// TIA Portal V18 export
DATA_BLOCK "CS_Drive_PL"   // DB10, Motion_DB
// stored: InstanceOfName TO_SynchronousAxis, OfSystemLibElement TO_SynchronousAxis, OfSystemLibVersion 7.0
TO_SynchronousAxis   // technology object, version 7.0
// stored: Connection Interface Actor, InputAddress 400, OutputAddress 400
// stored: Connection Interface Sensor[1], InputAddress 400, OutputAddress 400, SensorIndexInActorTelegram 1
   // // inherited from TO_PositioningAxis
   // // inherited from TO_SpeedAxis
   // // inherited from TO_Axis
   // // inherited from TO_Object
   // VAR
   //    Actor : TO_Struct_Actor;
   // END_VAR
   // VAR
   //    Sensor : Array[1..4] of TO_Struct_Sensor;
   //    PositionControl : TO_Struct_PositionControl;
   // END_VAR
   // VAR
   //    StatusSynchronizedMotion { ExternalWritable := 'False'; S7_SetPoint := 'True'} : TO_Struct_StatusSynchronizedMotion;
   // END_VAR
BEGIN
   Actor.Interface.AddressIn.RID := 16#208072a;
   Actor.Interface.AddressIn.AREA := 16#81;
   Actor.Interface.AddressIn.OFFSET := 400;
   Actor.Interface.AddressOut.RID := 16#208072b;
   Actor.Interface.AddressOut.AREA := 16#82;
   Actor.Interface.AddressOut.OFFSET := 400;
   Sensor[1].Interface.AddressIn.RID := 16#208072a;
   Sensor[1].Interface.AddressIn.AREA := 16#81;
   Sensor[1].Interface.AddressIn.OFFSET := 400;
   Sensor[1].Interface.AddressOut.RID := 16#208072b;
   Sensor[1].Interface.AddressOut.AREA := 16#82;
   Sensor[1].Interface.AddressOut.OFFSET := 400;
   PositionControl.EnableDSC := true;
   _Actor.Interface.Telegram := 105;
   _Sensor[1].Interface.Telegram := 105;
END_DATA_BLOCK
